FUNCTION F_ScalingByRef : BOOL
VAR_INPUT
	entireSensor : REFERENCE TO ST_Sensor;
END_VAR
VAR
END_VAR

IF entireSensor.rawTemp >=0 THEN
	entireSensor.scaledTemp := (entireSensor.rawTemp/327.67);
	F_ScalingByRef := TRUE;
	RETURN;
ELSE
	F_ScalingByRef:=FALSE;
	
END_IF

END_FUNCTION

(* stored: Version 1.1.0.1, ProductVersion 3.1.4024.12
   POU F_ScalingByRef: Id {06cb1697-cea5-4e69-b245-5af5ab9427a8}, SpecialFunc None *)
